PROGRAM MAIN
VAR
		
	nState: INT;
	sMsg	:	STRING :=	'Sistemde Hata Olustu	Hata Kodu	=	 ';
	sMsg2	: 	STRING;
	sVar	:	STRING;
		
	bSend	:	BOOL;
	bErr	:	BOOL;
	bBusy	:	BOOL;
	bExecute: BOOL;
	
	sAxis	:	ST_Axis;
	fbmail: FB_SmtpV3;
	fbMotion: FB_Motion;

	sMsg3: STRING;
	sVar2: STRING(255);
	F_TRIG1: F_TRIG;
	Sens1: BOOL;
	counter: INT;
END_VAR


fbMotion(Axis:= .Axis1 , StAxis:=sAxis);
ACT_System();

ACTION ACT_System:

	fbmail(
	sNetId:='192.168.48.1.1.1' , 
	sSmtpServer:='smtp.gmail.com' , 
	sUsername:= '*******@gmail.com', 
	sPassword:= '*********',         
	nEncryption:= 2,                 
	sFrom:= '********@gmail.com',    
	sTo:= '**********@gmail.com',    
	sCc:= , 
	sBcc:= , 
	sSubject:= 'Sistem Hatasi Mevcut', 
	pMessage:= , 
	cbMessage:= , 
	bExecute:=bSend , 
	tTimeout:=T#2S , 
	bBusy=>bBusy , 
	bError=>bErr , 
	nErrId=> );

	F_TRIG1(CLK:=Sens1 , Q=> );

	

	sMsg2	:=	UDINT_TO_STRING(axis2.NcToPlc.ErrorCode);
	sMsg3	:=	UDINT_TO_STRING(saxis.OUTPUT.bPowErrid);
	
	sVar	:=	CONCAT(STR1:=sMsg , STR2:=sMsg2 );
	sVar2	:=	CONCAT(STR1:=sMsg , STR2:=sMsg3 );
	
	sAxis.INPUT.fOverride	:=	100;
	sAxis.INPUT.bStop	:= FALSE;
	
CASE nState OF
	
	0:
	
		saxis.INPUT.bMoveAbs	:=	FALSE;

		IF  saxis.OUTPUT.bPowerActive
		AND NOT sAxis.OUTPUT.bAbsErr	
		AND saxis.OUTPUT.bPowerActive
		AND sAxis.OUTPUT.bPowerStat THEN
		 
			nState	:=	1;
						
		END_IF
		
	1:
				
		IF bExecute 
		AND NOT sAxis.OUTPUT.bPowerErr
		AND sAxis.OUTPUT.bPowerActive 
		AND NOT sAxis.OUTPUT.bStopActive THEN
		
			nState	:=	10;
		
		ELSIF sAxis.OUTPUT.bAbsErr THEN
			nState:=999;
		END_IF
		
	10:			
		sAxis.INPUT.bStop	:=	FALSE;
		sAxis.INPUT.bMoveAbs	:=	TRUE;
		sAxis.INPUT.fPosition	:= 10000;
		sAxis.INPUT.nVelocity	:=	5000;
		
		IF	sAxis.OUTPUT.bAbsBusy 
		AND NOT sAxis.OUTPUT.bPowerErr
		AND sAxis.OUTPUT.bPowerActive 
		AND NOT sAxis.OUTPUT.bStopActive THEN
					
			nState	:=	20;
				
		ELSIF sAxis.OUTPUT.bAbsErr THEN
			nState:=999;
		END_IF

	20:

		IF sAxis.OUTPUT.bAbsDone 
		AND NOT sAxis.OUTPUT.bPowerErr	
		AND NOT sAxis.OUTPUT.bAbsErr	
		AND saxis.OUTPUT.bPowerActive	THEN

			nState	:=	30;
			sAxis.INPUT.bMoveAbs	:=	FALSE;
				
		ELSIF sAxis.OUTPUT.bAbsErr THEN
			nState:=999;
		END_IF
			
	30:	
		sAxis.INPUT.bStop	:=	FALSE;
		sAxis.INPUT.bMoveAbs	:=	TRUE;
		sAxis.INPUT.fPosition	:= 45000;
		sAxis.INPUT.nVelocity	:=	7000;
			
		
		
			IF	sAxis.OUTPUT.bAbsBusy 
			AND NOT sAxis.OUTPUT.bPowerErr
			AND sAxis.OUTPUT.bPowerActive 
			AND NOT sAxis.OUTPUT.bStopActive THEN							
				nState	:=	40;		
			ELSIF sAxis.OUTPUT.bAbsErr THEN
				nState:=999;
			END_IF
	
				
	40:
		IF sAxis.OUTPUT.bAbsDone 
		AND NOT sAxis.OUTPUT.bPowerErr	
		AND NOT sAxis.OUTPUT.bAbsErr	
		AND saxis.OUTPUT.bPowerActive	THEN

		
			sAxis.INPUT.bMoveAbs	:=	FALSE;

			IF f_trig1.Q THEN
					
				counter	:=	counter	+	1;

				IF counter >=5 THEN
					counter	:=	0;
					nState	:=	50;
				END_IF
			
			END_IF

			
				
			ELSIF sAxis.OUTPUT.bAbsErr THEN
				nState:=999;
			END_IF
					
				
		50:	
			sAxis.INPUT.bStop	:=	FALSE;
			sAxis.INPUT.bMoveAbs	:=	TRUE;
			sAxis.INPUT.fPosition	:= 0;
			sAxis.INPUT.nVelocity	:=	7000;
		
			IF	sAxis.OUTPUT.bAbsBusy AND NOT	sAxis.OUTPUT.bPowerErr	
			AND NOT	sAxis.OUTPUT.bAbsErr	THEN
					
				nState	:=	60;
				
			ELSIF sAxis.OUTPUT.bAbsErr THEN
				nState:=999;
			END_IF
			
		60:

			IF sAxis.OUTPUT.bAbsDone AND NOT sAxis.OUTPUT.bPowerErr	
			AND NOT	sAxis.OUTPUT.bAbsErr	THEN

				nState	:=	0;
				sAxis.INPUT.bMoveAbs	:=	FALSE;
				
			ELSIF sAxis.OUTPUT.bAbsErr THEN
				nState:=999;
			END_IF
				
		999:
		
    	
			// Hataya neden olacak hata kodunu atacak şekilde düzenle
		
			saxis.INPUT.bReset	:=	TRUE;
			saxis.INPUT.bMoveAbs	:=	FALSE;
			
			fbmail.pMessage	:=	ADR(sVAr);
			fbmail.cbMessage	:=	SIZEOF(sVar);
			bSend	:=	TRUE;	
    		
		
			IF saxis.OUTPUT.bResetDone THEN
				nState	:=	1000;
			END_IF
			
		1000:
			
			IF NOT sAxis.OUTPUT.bPowerErr 
			AND NOT saxis.OUTPUT.bAbsErr
			AND saxis.OUTPUT.bPowerActive
			AND NOT saxis.OUTPUT.bPowerErr THEN
				
				bSend	:=	FALSE;
				nState	:=	0;
			
			END_IF
        	
	
END_CASE


	IF NOT bExecute THEN
		nState	:=	0;
		
		sAxis.INPUT.bStop	:=	TRUE;
		saxis.INPUT.bMoveAbs	:=	FALSE;
		
		sAxis.INPUT.fPosition	:= 0;
		sAxis.INPUT.nVelocity	:=	0;

			IF saxis.OUTPUT.bStopDone AND NOT sAxis.OUTPUT.bPowerErr 
			AND sAxis.OUTPUT.bPowerActive THEN
					sAxis.INPUT.bStop	:=	FALSE;
					nState	:=	0;
			END_IF
	END_IF

			
	
		IF 	saxis.OUTPUT.bPowerErr THEN
	
			fbmail.pMessage	:=	ADR(sVAr2);
			fbmail.cbMessage	:=	SIZEOF(sVar2);
			bSend	:=	TRUE;
		
			saxis.INPUT.bReset	:=	TRUE;
			
				IF saxis.OUTPUT.bResetDone 
				AND NOT saxis.OUTPUT.bAbsErr 
				AND NOT saxis.OUTPUT.bPowerErr THEN
					
					bSend	:=	FALSE;
					saxis.INPUT.bMoveAbs	:=	FALSE;
					nState	:=	0;
				
				END_IF
			END_IF
END_ACTION

END_PROGRAM

(* stored: Version 1.1.0.1, ProductVersion 3.1.4024.4
   POU MAIN: Id {bb863162-c9ea-4e78-b8ba-e4dff236f00d}, SpecialFunc None
   Action ACT_System: Id {285e1227-4524-48c2-8603-6f6e814b0bc0} *)
